FUNCTION_BLOCK FB_ForceMonitor

VAR_INPUT
	
	//Input parameters
    bEnable                  			:BOOL;   
    bActive                 			:BOOL;	//Monitoring active
	bReset								:BOOL;
    fForceInput              			:REAL;
    fThreshold_UpperLimit    			:REAL;
    fThreshold_LowerLimit   			:REAL;
	fDebounceTolerance   				:REAL;	// +/- range for stable
	fDistance							:REAL;
	fDisTanceSetPoint					:REAL;



END_VAR

VAR_OUTPUT
	
	//Output parameters
    bPass                  			    :BOOL;    //TRUE when within both limits
    bFail                    			:BOOL;    //TRUE if outside
    fHighestRecordedForce    			:REAL;
    fLowestRecordedForce     			:REAL;
    bOutOfRangeHigh          			:BOOL;
    bOutOfRangeLow           			:BOOL;
END_VAR

VAR
	//Debounce
	fForceInputABS						:REAL;

	tDebouncePeriod      				:TIME:= T#75MS;
	tonDebounce      					:Tc2_Standard.TON;
	fForceLastStable     				:REAL;
	fForceFiltered       				:REAL;
	bForceStable         				:BOOL;
	
	bDistancePass						:BOOL;
	//Logic support variables
    bActiveLast              			:BOOL;
    bEvaluate	             			:BOOL;
    bTracking                			:BOOL;
END_VAR

//----------------------------------------------------------------------oldschoo1

//Input ABS
IF fForceInput > 0 THEN      //Correct the error in negative read
fForceInputABS :=ABS(fForceInput);
ELSE 
	fForceInputABS:=0;
END_IF

// Transitions
bEvaluate 	:= NOT bActive AND bActiveLast;
bActiveLast := bActive;


// Debounce logic --------------------------------------------------------------*
IF (fForceInputABS - fForceLastStable) <= fDebounceTolerance THEN
    	tonDebounce(IN:=TRUE, PT:=tDebouncePeriod);
ELSE
    	tonDebounce(IN:=FALSE);
    	fForceLastStable:= fForceInputABS;
END_IF;

bForceStable := tonDebounce.Q;

IF bForceStable THEN fForceFiltered := fForceLastStable; END_IF


// LOGIC ------------------------------------------------------------------------*
IF bEnable  THEN

	//Record
    IF bActive THEN
					IF NOT bTracking THEN
						
						fHighestRecordedForce 	:= fForceInputABS;
						fLowestRecordedForce 	:= fForceInputABS;
						bTracking := TRUE;
						
					END_IF
						// Track max/min
					IF 	fDistance < fDisTanceSetPoint THEN
						IF fForceInputABS > fHighestRecordedForce THEN
							fHighestRecordedForce := fForceInputABS;
						END_IF;
			
						IF fForceInputABS < fLowestRecordedForce THEN
							fLowestRecordedForce  := fForceInputABS;
						END_IF;
					END_IF;
					
					
	//Evaluation
    ELSIF bEvaluate THEN
        
						bFail := (fHighestRecordedForce > fThreshold_UpperLimit) OR
      							 (fHighestRecordedForce  < fThreshold_LowerLimit);
						bPass := NOT bFail;
					
						bTracking := FALSE;
						bDistancePass := FALSE;					
    END_IF

ELSE
		// Clear 
		bPass 					:= FALSE;
		bFail 					:= FALSE;
		bOutOfRangeHigh 		:= FALSE;
		bOutOfRangeLow 			:= FALSE;
		fHighestRecordedForce 	:= 0.0;
		fLowestRecordedForce 	:= 0.0;
		bTracking 				:= FALSE;
		bActiveLast 			:= FALSE;
    	fForceLastStable 		:= 0.0;
    	fForceFiltered 			:= 0.0;
    	bForceStable 			:= FALSE;
		tonDebounce			 (IN:= FALSE);
END_IF

IF bReset THEN
		// Reset 
		bPass 					:= FALSE;
		bFail 					:= FALSE;
		bOutOfRangeHigh 		:= FALSE;
		bOutOfRangeLow 			:= FALSE;
		fHighestRecordedForce 	:= 0.0;
		fLowestRecordedForce 	:= 0.0;
		bTracking 				:= FALSE;
		bActiveLast 			:= FALSE;
    	fForceLastStable 		:= 0.0;
    	fForceFiltered 			:= 0.0;
    	bForceStable 			:= FALSE;
		tonDebounce			 (IN:= FALSE);
END_IF
//----------------------------------------------------------------------------oldschoo1

END_FUNCTION_BLOCK

(* stored: Version 1.1.0.1, ProductVersion 3.1.4024.13
   POU FB_ForceMonitor: Id {78deaf87-f7b5-4af9-bf4d-a4d57928b991}, SpecialFunc None *)
